// TIA Portal V17 export
// export: Created 2021-12-03T08:13:09.5263887Z, ExportSetting WithDefaults, DisplayName Totally Integrated Automation Portal, DisplayVersion V17, DisplayName TIA Portal Openness, DisplayVersion V17, DisplayName TIA Portal Version Control Interface, DisplayVersion V17, DisplayName STEP 7 Professional, DisplayVersion V17, DisplayName STEP 7 Safety, DisplayVersion V17, DisplayName WinCC Advanced, DisplayVersion V17
ORGANIZATION_BLOCK "CYC_INT4_RTG1"   // OB34, STL, CyclicInterrupt
TITLE = "Cyclic Interrupt"
VERSION : 0.1
   VAR_TEMP
      OB34_EV_CLASS : Byte;   // Bits 0-3 = 1 (Coming event), Bits 4-7 = 1 (Event class 1)
      OB34_STRT_INF : Byte;   // 16#35 (OB 34 has started)
      OB34_PRIORITY : Byte;   // Priority of OB Execution
      OB34_OB_NUMBR : Byte;   // 34 (Organization block 34, OB34)
      OB34_RESERVED_1 : Byte;   // Reserved for system
      OB34_RESERVED_2 : Byte;   // Reserved for system
      OB34_PHS_OFFSET : Int;   // Phase offset (integer, milliseconds)
      OB34_RESERVED_3 : Int;   // Reserved for system
      OB34_EXC_FREQ : Int;   // Frequency of execution (msec)
      OB34_DATE_TIME : Date_And_Time;   // Date and time OB34 started
   END_VAR
BEGIN

NETWORK
TITLE = 

      CALL  "Main_Safety_RTG1", "FDBI_Main_Safety_RTG11";
      NOP   0;
END_ORGANIZATION_BLOCK
